FUNCTION Convert_LREAL_TO_LREAL : BOOL
VAR_INPUT
	in : LREAL;
	out : REFERENCE TO LREAL;
END_VAR

out := in;
Convert_LREAL_TO_LREAL := TRUE;

END_FUNCTION

(* stored: Version 1.1.0.1, ProductVersion 3.1.4024.12
   POU Convert_LREAL_TO_LREAL: Id {2f9269b1-4893-4977-9a61-5aa919f2bebb}, SpecialFunc None *)
